Fanuc KAREL source: kb00166.KL

-- PROVISIONAL review KL for V770-1; original PC SHA256 8d8421bd083a8af02fa833d90fb6c90819f19f9c9323c4b7103ceab0712d755f
-- Incomplete behavior may be omitted. Consult companion uncertainty JSON. Do not deploy.
PROGRAM KB00166
%NOLOCKGROUP
BEGIN
  -- UNRESOLVED_PC offsets 5-12; opcodes 9D,23
  -- UNRESOLVED_PC offsets 17-24; opcodes 9D,23
  -- UNRESOLVED_PC offsets 29-59; opcodes 27,22,22,1C,22,27,9D,31
  -- UNRESOLVED_PC offsets 64-68; opcodes 7F
END KB00166
